{attribute 'qualified_only'}
{attribute 'strict'}
TYPE E_SwitchOpMode :
(
  Blend         := 0,
  WithoutSwitch := 1,
  SwitchOnly    := 2
);
END_TYPE

(* stored: Version 1.1.0.1
   DUT E_SwitchOpMode: Id {336cc65d-a64d-0f73-1268-f248dcfeb0a0} *)
